// TIA Portal V20 export
TYPE "typeCutCount"
// stored: Access Published, Namespace Unit1.Em7
   STRUCT
      cutCountPV : DInt;
      cutCountLimitWarningSV : DInt;
      cutCountLimitAlarmSV : DInt;
      cutCountReset : Bool;
   END_STRUCT;
END_TYPE
